FUNCTION_BLOCK Coche
VAR_INPUT 
END_VAR
VAR_OUTPUT
END_VAR
VAR_IN_OUT
END_VAR
VAR
	_Marca : STRING;
	_Color : STRING;
	accion : STRING;
END_VAR

METHOD PUBLIC Acelerar
accion := 'acelerar';
END_METHOD

PROPERTY PUBLIC Color : STRING
GET
Color := _Color;
END_GET
SET
_Color := Color;
END_SET
END_PROPERTY

METHOD PUBLIC Conducir
accion := 'conducir';
END_METHOD

METHOD PUBLIC Frenar
accion := 'frenar';
END_METHOD

PROPERTY PUBLIC Marca : STRING
GET
Marca := _Marca;
END_GET
SET
_Marca := Marca;
END_SET
END_PROPERTY

END_FUNCTION_BLOCK

(* stored: Version 1.1.0.1, ProductVersion 3.1.4024.12
   POU Coche: Id {d772e4a1-e405-4c42-bf3e-790247ec68f4}, SpecialFunc None
   Folder Metodos: Id {e93741ea-181a-4006-8f66-9dfbb29cf23b}
   Folder Propiedades: Id {a3aa27d7-8148-4244-88cb-ee03d1f6c74c}
   Method Acelerar: Id {df6cf032-d981-4328-a5c3-ffc2361c2bc9}
   Property Color: Id {aa2c479c-72b5-4532-9433-83f1084fe047}
   Get Get: Id {43ad63d7-5b92-45bd-8b4e-2c01e4811dfb}
   Set Set: Id {2ed5c4f3-57ec-4058-adc5-6c141ced88d5}
   Method Conducir: Id {5067b8ca-bfa3-44a9-8fb6-c937f24afb9f}
   Method Frenar: Id {c4768733-2c2f-4f12-8d0a-d6df21d35961}
   Property Marca: Id {0f522775-9d24-483d-a844-018bfeb11cb7}
   Get Get: Id {0f63c98c-c8c3-4246-8e7a-9eb79d0d3e90}
   Set Set: Id {cc521b98-57fd-4b78-902f-6015af7cbf49} *)
